TYPE CmpConvStop :
STRUCT
	Framework: Framework;
	Available: BOOL;
	Release: BOOL;
	WorkReq: BOOL;
	WorkCmp: BOOL;
	ConvRunning: BOOL;
	StatusInCycleAuto: BOOL;
	StatusPuckPresent: BOOL;
	StatusBufferFull: BOOL;
	RemoteBufferFull: BOOL;
	FreeRunCycleStop: BOOL;
	Config: CmpConvStopConfig;
END_STRUCT
END_TYPE

(* stored: Version 1.1.0.1, ProductVersion 3.1.4024.6
   DUT CmpConvStop: Id {d96649ef-31cf-4294-b860-eb238cd627cb} *)
